(* IEC 61131-3 sources: SMRamp/src/Ar/SMRamp, 21 files *)

(* ---- SMRamp.typ ---- *)
(*
* File: SMRamp.typ
* Copyright (c) 2023 Loupe
* https://loupe.team
*
* This file is part of SMRamp, licensed under the MIT License.
*
*)

TYPE
	SMR_Axis_Int_ParUpdate_typ : 	STRUCT
		Update : BOOL;
		CurrValue : UINT;
		AccWrite : AsIOAccWrite;
	END_STRUCT;
	SMR_Axis_Int_Homing_typ : 	STRUCT
		State : UINT;
		CurrDirection : SINT; (*Current direction of travel*)
		HomeSwOld : BOOL; (*Previous value of HomeSw input for edge detection*)
		RisingEdge : BOOL; (*A rising edge was detected (not dependent on direction of travel)*)
		FallingEdge : BOOL; (*A falling edge was detected (not dependent on direction of travel)*)
		PosEdge : BOOL; (*A "Positive" edge was detected (depends on direction of travel)*)
		NegEdge : BOOL; (*A "Negative" edge was detected (depends on direction of travel)*)
		PosLimitSwOld : BOOL; (*Previous value of PosLimitSw for edge detection*)
		PosLimitSwRisingEdge : BOOL; (*An edge was detected for the PosLimitSw*)
		PosLimitSwFallingEdge : BOOL; (*An edge was detected for the PosLimitSw*)
		NegLimitSwOld : BOOL; (*Previous value of NegLimitSw for edge detection*)
		NegLimitSwRisingEdge : BOOL; (*An edge was detected for the NegLimitSw*)
		NegLimitSwFallingEdge : BOOL; (*An edge was detected for the NegLimitSw*)
		TargetReachedTimer : TON; (*Timer to ensure that TargetReached is true for long enough (takes care of timing issues, but makes homing slightly slower (100-200ms)).*)
	END_STRUCT;
	SMR_Axis_Internal_typ : 	STRUCT
		CMD : SMR_Axis_IN_CMD_typ; (*Internal CMD structure for discriminating between new and old commands.*)
		DIGIN : SMR_Axis_IOMap_IN_typ; (*Holds logical values of digital inputs (for future expansion)*)
		AbsPos : DINT;
		AbsPosActVal : DINT;
		CurrTargetPos : DINT;
		CurrTargetVel : DINT;
		CurrDirection : SINT;
		EnableState : UINT;
		SetState : UINT;
		Error : BOOL; (*Internal code error*)
		TargetReachedTimer : TON; (*Timer to ensure that TargetReached is true for long enough. Used to set Busy and Done in velocity mode.*)
		AckResetTimer : TON; (*Timer to ensure that the hardware fault acknowledge bits are high for long enough to be seen*)
		Homing : SMR_Axis_Int_Homing_typ;
		UpdateVel : SMR_Axis_Int_ParUpdate_typ;
		UpdateAcc : SMR_Axis_Int_ParUpdate_typ;
		UpdateDec : SMR_Axis_Int_ParUpdate_typ;
		ParsOK : BOOL; (*All motion parameters are up to date*)
		RTInfo : RTInfo; (*RTInfo block to get cycle time*)
		SpdEst : SpeedEst; (*SpdEst block to estimate speed*)
	END_STRUCT;
	SMR_Axis_IOMap_OUT_typ : 	STRUCT
		AbsPos : DINT;
		MpGenControl : UINT;
		MpGenMode : SINT;
	END_STRUCT;
	SMR_Axis_IOMap_IN_typ : 	STRUCT
		HomeSw : BOOL;
		PosLimitSw : BOOL;
		NegLimitSw : BOOL;
		QuickStop : BOOL;
		AbsPosActVal : DINT;
		MpGenStatus : UINT;
	END_STRUCT;
	SMR_Axis_IOMap_typ : 	STRUCT
		IN : SMR_Axis_IOMap_IN_typ;
		OUT : SMR_Axis_IOMap_OUT_typ;
	END_STRUCT;
	SMR_Axis_TEST_STAT_typ : 	STRUCT
		Busy : BOOL;
		Done : BOOL;
		Error : BOOL; (*Motor Fault or InternalError exists*)
		ErrorID : UINT;
		ErrorString : STRING[SMR_STRLEN_ERROR];
		ActualPosition : DINT;
		ActualVelocity : REAL; (*NOT IMPLEMENTED YET*)
		State : UINT;
		DriveFault : BOOL;
		VoltageEnabled : BOOL;
		HomingOk : BOOL;
	END_STRUCT;
	SMR_Axis_TEST_typ : 	STRUCT
		Enable : BOOL;
		CMD : SMR_Axis_IN_CMD_typ;
		PAR : SMR_Axis_IN_PAR_typ;
		STAT : SMR_Axis_TEST_STAT_typ;
	END_STRUCT;
	SMR_Axis_OUT_STAT_DriveStat_typ : 	STRUCT
		RdyToSwOn : BOOL;
		SwOn : BOOL;
		OpEnabled : BOOL;
		Fault : BOOL;
		VoltageEnabled : BOOL;
		QuickStop : BOOL;
		SwOnDisabled : BOOL;
		Warning : BOOL;
		Remote : BOOL;
		TargetReached : BOOL;
		IntLimitActive : BOOL;
		MotorLoad0 : BOOL;
		MotorLoad1 : BOOL;
		MotorLoad2 : BOOL;
		HomingOk : BOOL;
	END_STRUCT;
	SMR_Axis_OUT_STAT_typ : 	STRUCT
		ReadyForCMD : BOOL;
		Busy : BOOL;
		Done : BOOL;
		Error : BOOL; (*Motor Fault or InternalError exists*)
		ErrorID : UINT;
		ErrorString : STRING[SMR_STRLEN_ERROR];
		ErrorState : UINT;
		ActualPosition : DINT;
		ActualVelocity : REAL; (*Velocity in usteps/s or cts/s, depending on IN.CFG.ABRCtrSyncAsync. THIS WILL NOT MATCH VELOCITY INPUT BECAUSE OF DIFFERENT UNITS.*)
		DriveStatus : SMR_Axis_OUT_STAT_DriveStat_typ;
		State : UINT;
	END_STRUCT;
	SMR_Axis_OUT_typ : 	STRUCT
		STAT : SMR_Axis_OUT_STAT_typ;
	END_STRUCT;
	SMR_Axis_IN_CFG_SpdEst_typ : 	STRUCT
		tf : REAL;
		deadband : DINT;
		K : REAL;
	END_STRUCT;
	SMR_Axis_IN_CFG_typ : 	STRUCT
		DisableAcyclicWrite : BOOL;
		ModuleINADeviceName : STRING[80];
		MotorIndex : USINT;
		UnderCurrentDetection : BOOL;
		ABRCtrSyncAsync : BOOL;
		StallDetection : BOOL;
		InvertDirection : BOOL;
		SpeedEstimator : SMR_Axis_IN_CFG_SpdEst_typ;
	END_STRUCT;
	SMR_Axis_IN_PAR_typ : 	STRUCT
		HomingPosition : DINT;
		HomingMode : SINT;
		HomingVelocity : UINT;
		HomingStartDir : SINT;
		HomingEdgeSw : SINT;
		HomingTriggDir : SINT;
		Position : DINT;
		Direction : SINT;
		Velocity : UINT;
		Acceleration : UINT;
		Deceleration : UINT;
		JogVelocity : UINT;
		StopDeceleration : UINT;
	END_STRUCT;
	SMR_Axis_IN_CMD_typ : 	STRUCT
		Power : BOOL;
		Home : BOOL;
		MoveAbsolute : BOOL;
		MoveAdditive : BOOL;
		MoveVelocity : BOOL;
		JogForward : BOOL;
		JogReverse : BOOL;
		TrackSetPosition : BOOL;
		Stop : BOOL;
		AcknowledgeError : BOOL;
	END_STRUCT;
	SMR_Axis_IN_typ : 	STRUCT
		CMD : SMR_Axis_IN_CMD_typ;
		PAR : SMR_Axis_IN_PAR_typ;
		CFG : SMR_Axis_IN_CFG_typ;
	END_STRUCT;
	SMR_Axis_typ : 	STRUCT
		IN : SMR_Axis_IN_typ;
		OUT : SMR_Axis_OUT_typ;
		TEST : SMR_Axis_TEST_typ;
		IOMap : SMR_Axis_IOMap_typ;
		Internal : SMR_Axis_Internal_typ;
	END_STRUCT;
END_TYPE

(* ---- SMR_CheckHomePAR.st ---- *)
(*
* File: SMR_CheckHomePAR.st
* Copyright (c) 2023 Loupe
* https://loupe.team
*
* This file is part of SMRamp, licensed under the MIT License.
*
*)

(*Function which checks homing parameters.  Returns TRUE if pars are OK.*)

(* Parameter checking			DONE and TESTED DFB 20090914 *)

FUNCTION SMR_CheckHomePAR

(* Reset internal Error variable.  Will be set below if there is an error *)

Error:=	0;

(* Check HomingMode *)

IF( 	(pAxis.IN.PAR.HomingMode <> SMR_HOMEMODE_DIRECT)
	AND (pAxis.IN.PAR.HomingMode <> SMR_HOMEMODE_SWITCH_GATE)
	AND	(pAxis.IN.PAR.HomingMode <> SMR_HOMEMODE_ABS_SWITCH)
	AND	(pAxis.IN.PAR.HomingMode <> SMR_HOMEMODE_END_SWITCH)
	)THEN

 	Error:=	1;

END_IF

(* Check HomingVelocity *)

IF( pAxis.IN.PAR.HomingVelocity = 0 )THEN

 	Error:=	1;

END_IF

(* Check HomingStartDir *)

IF( 	(pAxis.IN.PAR.HomingStartDir <> SMR_POS)
	AND (pAxis.IN.PAR.HomingStartDir <> SMR_NEG)
	)THEN

 	Error:=	1;

END_IF

(* Check HomingEdgeSw *)

IF( 	(pAxis.IN.PAR.HomingEdgeSw <> SMR_POS)
	AND	(pAxis.IN.PAR.HomingEdgeSw <> SMR_NEG)
	)THEN

 	Error:=	1;

END_IF

(* Check HomingTriggDir *)

IF( 	(pAxis.IN.PAR.HomingTriggDir <> SMR_POS)
	AND	(pAxis.IN.PAR.HomingTriggDir <> SMR_NEG)
	)THEN

 	Error:=	1;

END_IF

IF( Error )THEN

	SMR_CheckHomePAR:=	0;

ELSE

	SMR_CheckHomePAR:=	1;

END_IF

END_FUNCTION

(* ---- SMR_CheckLimitSw.st ---- *)
(*
* File: SMR_CheckLimitSw.st
* Copyright (c) 2023 Loupe
* https://loupe.team
*
* This file is part of SMRamp, licensed under the MIT License.
*
*)

(********************************************************************)
(* Check limit switches 											*)
(********************************************************************)

FUNCTION SMR_CheckLimitSw

(********************************************************************)
(* Set return value to get rid of compiler warning					*)
(********************************************************************)

SMR_CheckLimitSw:=	FALSE;

(********************************************************************)
(* Check Limit Switches												*)
(********************************************************************)

(* PosLimitSw *)

IF( (pAxis.Internal.CurrDirection = SMR_DIR_POS)
	AND	(pAxis.Internal.DIGIN.PosLimitSw)
	)THEN

	(* Set CurrDirection to STOP *)

	pAxis.Internal.CurrDirection:=	SMR_DIR_STOP;

	(* Set Mode to Velocity mode and set position to 0 to stop axis *)

	pAxis.IOMap.OUT.MpGenMode:=	SMR_MODE_VELOCITY;
	pAxis.Internal.AbsPos:=		0;

	(* Set Error info and go to Error state *)

	pAxis.Internal.Error:=			1;
	pAxis.OUT.STAT.ErrorID:=		SMR_ERR_POSLIMSW;
	pAxis.OUT.STAT.ErrorState:=		pAxis.Internal.EnableState;

	pAxis.Internal.EnableState:=	SMR_STEN_ERROR;

	(* Reset Busy and Done *)

	pAxis.OUT.STAT.Busy:=	0;
	pAxis.OUT.STAT.Done:=	0;

END_IF

(* NegLimitSw *)

IF( (pAxis.Internal.CurrDirection = SMR_DIR_NEG)
	AND	(pAxis.Internal.DIGIN.NegLimitSw)
	)THEN

	(* Set CurrDirection to STOP *)

	pAxis.Internal.CurrDirection:=	SMR_DIR_STOP;

	(* Set Mode to Velocity mode and set position to 0 to stop axis *)

	pAxis.IOMap.OUT.MpGenMode:=	SMR_MODE_VELOCITY;
	pAxis.Internal.AbsPos:=		0;

	(* Set Error info and go to Error state *)

	pAxis.Internal.Error:=			1;
	pAxis.OUT.STAT.ErrorID:=		SMR_ERR_NEGLIMSW;
	pAxis.OUT.STAT.ErrorState:=		pAxis.Internal.EnableState;

	pAxis.Internal.EnableState:=	SMR_STEN_ERROR;

	(* Reset Busy and Done *)

	pAxis.OUT.STAT.Busy:=	0;
	pAxis.OUT.STAT.Done:=	0;

END_IF

END_FUNCTION

(* ---- SMR_GetDriveStatus.st ---- *)
(*
* File: SMR_GetDriveStatus.st
* Copyright (c) 2023 Loupe
* https://loupe.team
*
* This file is part of SMRamp, licensed under the MIT License.
*
*)

(*This is an internal function that maps out the status from the status UINT.*)

(* Getting status			DONE and TESTED DFB 20110329 *)

FUNCTION SMR_GetDriveStatus

(********************************************************************)
(* Set return value to get rid of compiler warning					*)
(********************************************************************)

SMR_GetDriveStatus:=	FALSE;

(* Get status BOOLs out of status UINT *)

DriveStatus.RdyToSwOn:=			BIT_TST(MpGenStatus, 0);
DriveStatus.SwOn:=				BIT_TST(MpGenStatus, 1);
DriveStatus.OpEnabled:=			BIT_TST(MpGenStatus, 2);
DriveStatus.Fault:=				BIT_TST(MpGenStatus, 3);
DriveStatus.VoltageEnabled:=	BIT_TST(MpGenStatus, 4);
DriveStatus.QuickStop:=			BIT_TST(MpGenStatus, 5);
DriveStatus.SwOnDisabled:=		BIT_TST(MpGenStatus, 6);
DriveStatus.Warning:=			BIT_TST(MpGenStatus, 7);

DriveStatus.Remote:=			BIT_TST(MpGenStatus, 9);
DriveStatus.TargetReached:=		BIT_TST(MpGenStatus, 10);
DriveStatus.IntLimitActive:=	BIT_TST(MpGenStatus, 11);

DriveStatus.MotorLoad0:=		BIT_TST(MpGenStatus, 13);
DriveStatus.MotorLoad1:=		BIT_TST(MpGenStatus, 14);
DriveStatus.MotorLoad2:=		BIT_TST(MpGenStatus, 15);

END_FUNCTION

(* ---- SMR_Home.st ---- *)
(*
* File: SMR_Home.st
* Copyright (c) 2023 Loupe
* https://loupe.team
*
* This file is part of SMRamp, licensed under the MIT License.
*
*)

(*Function to perform homing functionality.*)

(* Stop during home										DONE and TESTED DFB 20110404 *)
	(* Setting SetState									DONE and TESTED DFB 20110404 *)
	(* Changing State									DONE and TESTED DFB 20110404 *)

(* Checking parameters									see CheckHomePAR.st *)
	(* Finding bad parameters							see CheckHomePAR.st *)
	(* Reacting to bad parameters						DONE and TESTED DFB 20090918 *)

(* Finding events										see HomeFindEdge.st *)

(* Starting Homing - change state based on mode			DONE and TESTED DFB 20090918 *)

(* Homing Modes											DONE and TESTED DFB 20090921 *)

	(* Direct											DONE and TESTED DFB 20090918 *)

	(* Switch gate mode									DONE and TESTED DFB 20090918 *)

		(* StartDir = Positive							DONE and TESTED DFB 20090918 *)

			(* EdgeSw = Positive						DONE and TESTED DFB 20090918 *)
				(* TriggDir = Positive					DONE and TESTED DFB 20090918 *)
				(* TriggDir = Negative					DONE and TESTED DFB 20090918 *)

			(* EdgeSw = Negative						DONE and TESTED DFB 20090918 *)
				(* TriggDir = Positive					DONE and TESTED DFB 20090918 *)
				(* TriggDir = Negative					DONE and TESTED DFB 20090918 *)

		(* StartDir = Negative							DONE and TESTED DFB 20090918 *)

			(* EdgeSw = Positive						DONE and TESTED DFB 20090918 *)
				(* TriggDir = Positive					DONE and TESTED DFB 20090918 *)
				(* TriggDir = Negative					DONE and TESTED DFB 20090918 *)

			(* EdgeSw = Negative						DONE and TESTED DFB 20090918 *)
				(* TriggDir = Positive					DONE and TESTED DFB 20090918 *)
				(* TriggDir = Negative					DONE and TESTED DFB 20090918 *)

	(* Abs Switch mode									DONE and TESTED DFB 20090918 *)

		(* EdgeSw = Positive							DONE and TESTED DFB 20090918 *)
			(* TriggDir = Positive						DONE and TESTED DFB 20090918 *)
			(* TriggDir = Negative						DONE and TESTED DFB 20090918 *)

		(* EdgeSw = Negative							DONE and TESTED DFB 20090918 *)
			(* TriggDir = Positive						DONE and TESTED DFB 20090918 *)
			(* TriggDir = Negative						DONE and TESTED DFB 20090918 *)

	(* End switch										DONE and TESTED DFB 20090921 *)

		(* EdgeSw = Positive							DONE and TESTED DFB 20090921 *)
			(* TriggDir = Positive						DONE and TESTED DFB 20090921 *)
			(* TriggDir = Negative						DONE and TESTED DFB 20090921 *)

		(* EdgeSw = Negative							DONE and TESTED DFB 20090921 *)
			(* TriggDir = Positive						DONE and TESTED DFB 20090921 *)
			(* TriggDir = Negative						DONE and TESTED DFB 20090921 *)

(* Finishing homing										DONE and TESTED DFB 20090918 *)

	(* Setting ActPos to HomeOffset						DONE and TESTED DFB 20090918 *)
		(* Mode and AbsPos setting						DONE and TESTED DFB 20110906 *)

	(* Timing on TargetReached							DONE and TESTED DFB 20090918 *)
		(* 5ms TC										DONE and TESTED DFB 20090918 *)
		(* 25ms TC										DONE and TESTED DFB 20090918 *)
		(* 50ms TC										DONE and TESTED DFB 20090918 *)

	(* Being at HomeOffset after homing					DONE and TESTED DFB 20090918 *)
		(* Mode and AbsPos setting						DONE and TESTED DFB 20110906 *)

	(* Setting HomingComplete 							DONE and TESTED DFB 20090918 *)

FUNCTION SMR_Home

(********************************************************************)
(* Set return value to get rid of compiler warning					*)
(********************************************************************)

SMR_Home:=	FALSE;

(* Map pointer to internal homing variables *)

t ACCESS ADR(pAxis.Internal.Homing);

(********************************************************************)
(* Reset TargetReachedTimer.  It will be set below when appropriate	*)
(********************************************************************)

t.TargetReachedTimer.IN:=	0;

(********************************************************************)
(* Stop command can interrupt a home move 							*)
(********************************************************************)

IF( pAxis.IN.CMD.Stop ) THEN

	(* Set the target state as SETSTOP *)

	pAxis.Internal.SetState:=		SMR_STEN_SETSTOP;

	(* Set Busy, Done *)

	pAxis.OUT.STAT.Busy:=	1;
	pAxis.OUT.STAT.Done:=	0;

	(* Go to SetState *)

	pAxis.Internal.EnableState:=	pAxis.Internal.SetState;

	RETURN;

END_IF

(********************************************************************)
(* Check Homing Parameters											*)
(********************************************************************)

IF( SMR_CheckHomePAR( pAxis ) = FALSE ) THEN

	(* Error - set internal error and go to error state *)

	pAxis.Internal.Error:=			1;
	pAxis.OUT.STAT.ErrorID:=		SMR_ERR_HOME_INVALIDPAR;
	pAxis.OUT.STAT.ErrorState:=		pAxis.Internal.EnableState;

	pAxis.Internal.EnableState:=	SMR_STEN_ERROR;

	RETURN;

END_IF

(********************************************************************)
(* Find edges 														*)
(********************************************************************)

SMR_HomeFindEdge( pAxis );

(********************************************************************)
(* Main State Machine												*)
(********************************************************************)

CASE t.State OF

	(********************************************************************)
	(* Starting Homing													*)
	(********************************************************************)

	SMR_STHOME_CHECKMODE:

		(* Stop motor when homing is initiated *)

		pAxis.IOMap.OUT.MpGenMode:=	SMR_MODE_VELOCITY;
		pAxis.Internal.AbsPos:=		0;

		(* Change state based on homing mode *)

		IF( pAxis.IN.PAR.HomingMode = SMR_HOMEMODE_DIRECT ) THEN

			(* If direct home, set homeoffset directly after motor is stopped *)

			t.State:=	SMR_STHOME_STOPPING;

  		ELSIF( pAxis.IN.PAR.HomingMode = SMR_HOMEMODE_SWITCH_GATE ) THEN

			t.State:=	SMR_STHOME_SG_START;

  		ELSIF( pAxis.IN.PAR.HomingMode = SMR_HOMEMODE_ABS_SWITCH ) THEN

			t.State:=	SMR_STHOME_ABS_START;

  		ELSIF( pAxis.IN.PAR.HomingMode = SMR_HOMEMODE_END_SWITCH ) THEN

			t.State:=	SMR_STHOME_END_START;

		END_IF

	(********************************************************************)
	(* Switch Gate mode													*)
	(********************************************************************)

	SMR_STHOME_SG_START:

		IF( pAxis.IN.PAR.HomingStartDir = SMR_POS ) THEN

			IF( pAxis.Internal.DIGIN.PosLimitSw ) THEN

   				t.CurrDirection:=	SMR_DIR_NEG;

			ELSE

				t.CurrDirection:=	SMR_DIR_POS;

			END_IF

		ELSIF( pAxis.IN.PAR.HomingStartDir = SMR_NEG ) THEN

			IF( pAxis.Internal.DIGIN.NegLimitSw ) THEN

   				t.CurrDirection:=	SMR_DIR_POS;

			ELSE

				t.CurrDirection:=	SMR_DIR_NEG;

			END_IF

		END_IF

		(* Change state *)

		t.State:=	SMR_STHOME_SG_MOVE;

		(* Set mode and velocity *)

		pAxis.IOMap.OUT.MpGenMode:=	SMR_MODE_VELOCITY;
		pAxis.Internal.AbsPos:=		UINT_TO_DINT(pAxis.IN.PAR.HomingVelocity) * t.CurrDirection;

	SMR_STHOME_SG_MOVE:

		(* Check all possible events and react accordingly *)

		(****************************************************)
		(* NegLimitSw *)

		IF( pAxis.Internal.DIGIN.NegLimitSw ) THEN

			(************************************************)
			(* NegLimitSw, NegDir *)

			IF( t.CurrDirection = SMR_DIR_NEG ) THEN

   				IF( pAxis.IN.PAR.HomingStartDir = SMR_POS ) THEN

					(* Stop, error *)

					t.CurrDirection:=	SMR_DIR_STOP;

					pAxis.Internal.Error:=			1;
					pAxis.OUT.STAT.ErrorID:=		SMR_ERR_HOME_ERR;
					pAxis.OUT.STAT.ErrorState:=		pAxis.Internal.EnableState;

					pAxis.Internal.EnableState:=	SMR_STEN_ERROR;

	   			ELSIF( pAxis.IN.PAR.HomingStartDir = SMR_NEG ) THEN

					(* Turn around to look for switch *)

					t.CurrDirection:=	SMR_DIR_POS;

				END_IF (* HomeStartDir *)

   			END_IF (* CurrDirection *)

		(****************************************************)
		(* PosLimitSw *)

		ELSIF( pAxis.Internal.DIGIN.PosLimitSw ) THEN

			(************************************************)
			(* PosLimitSw, PosDir *)

			IF( t.CurrDirection = SMR_DIR_POS ) THEN

				IF( pAxis.IN.PAR.HomingStartDir = SMR_POS ) THEN

					(* Turn around to look for switch *)

					t.CurrDirection:=	SMR_DIR_NEG;

	   			ELSIF( pAxis.IN.PAR.HomingStartDir = SMR_NEG ) THEN

					(* Stop, error *)

					t.CurrDirection:=	SMR_DIR_STOP;

					pAxis.Internal.Error:=			1;
					pAxis.OUT.STAT.ErrorID:=		SMR_ERR_HOME_ERR;
					pAxis.OUT.STAT.ErrorState:=		pAxis.Internal.EnableState;

					pAxis.Internal.EnableState:=	SMR_STEN_ERROR;

				END_IF (* HomeStartDir *)

			END_IF (* CurrDirection *)

		(****************************************************)
		(* PosEdge *)

		ELSIF( t.PosEdge ) THEN

  			(************************************************)
			(* PosEdge, PosDir *)

			IF( t.CurrDirection = SMR_DIR_POS ) THEN

				IF( pAxis.IN.PAR.HomingEdgeSw = SMR_POS ) THEN

					IF( pAxis.IN.PAR.HomingTriggDir = SMR_POS ) THEN

						(* Stop, done *)

						t.CurrDirection:=	SMR_DIR_STOP;

						t.State:=			SMR_STHOME_STOPPING;

	 				ELSIF( pAxis.IN.PAR.HomingTriggDir = SMR_NEG ) THEN

						(* Go negative *)

						t.CurrDirection:=	SMR_DIR_NEG;

	 				END_IF (* HomeTriggDir *)

				ELSIF( pAxis.IN.PAR.HomingEdgeSw = SMR_NEG ) THEN

					(* Find negative edge *)

					t.CurrDirection:=	SMR_DIR_POS;

				END_IF (* HomeEdgeSw *)

   			(************************************************)
			(* PosEdge, NegDir *)

			ELSIF( t.CurrDirection = SMR_DIR_NEG ) THEN

				IF( pAxis.IN.PAR.HomingEdgeSw = SMR_POS ) THEN

					IF( pAxis.IN.PAR.HomingTriggDir = SMR_POS ) THEN

						(* Go positive *)

						t.CurrDirection:=	SMR_DIR_POS;

	 				ELSIF( pAxis.IN.PAR.HomingTriggDir = SMR_NEG ) THEN

						(* Stop, done *)

						t.CurrDirection:=	SMR_DIR_STOP;

						t.State:=			SMR_STHOME_STOPPING;

	 				END_IF (* HomeTriggDir *)

				ELSIF( pAxis.IN.PAR.HomingEdgeSw = SMR_NEG ) THEN

					(* Find negative edge *)

					t.CurrDirection:=	SMR_DIR_POS;

				END_IF (* HomeEdgeSw *)

   			END_IF (* CurrDirection *)

		(****************************************************)
		(* NegEdge *)

  		ELSIF( t.NegEdge ) THEN

  			(************************************************)
			(* NegEdge, PosDir *)

			IF( t.CurrDirection = SMR_DIR_POS ) THEN

				IF( pAxis.IN.PAR.HomingEdgeSw = SMR_POS ) THEN

					(* Find positive edge *)

					t.CurrDirection:=	SMR_DIR_NEG;

				ELSIF( pAxis.IN.PAR.HomingEdgeSw = SMR_NEG ) THEN

					IF( pAxis.IN.PAR.HomingTriggDir = SMR_POS ) THEN

						(* Stop, done *)

						t.CurrDirection:=	SMR_DIR_STOP;

						t.State:=			SMR_STHOME_STOPPING;

	 				ELSIF( pAxis.IN.PAR.HomingTriggDir = SMR_NEG ) THEN

						(* Go negative *)

						t.CurrDirection:=	SMR_DIR_NEG;

	 				END_IF (* HomeTriggDir *)

				END_IF (* HomeEdgeSw *)

   			(************************************************)
			(* NegEdge, NegDir *)

			ELSIF( t.CurrDirection = SMR_DIR_NEG ) THEN

				IF( pAxis.IN.PAR.HomingEdgeSw = SMR_POS ) THEN

					(* Find positive edge *)

					t.CurrDirection:=	SMR_DIR_NEG;

				ELSIF( pAxis.IN.PAR.HomingEdgeSw = SMR_NEG ) THEN

					IF( pAxis.IN.PAR.HomingTriggDir = SMR_POS ) THEN

						(* Go positive *)

						t.CurrDirection:=	SMR_DIR_POS;

	 				ELSIF( pAxis.IN.PAR.HomingTriggDir = SMR_NEG ) THEN

						(* Stop, done *)

						t.CurrDirection:=	SMR_DIR_STOP;

						t.State:=			SMR_STHOME_STOPPING;

	 				END_IF (* HomeTriggDir *)

				END_IF (* HomeEdgeSw *)

   			END_IF (* CurrDirection *)

  		END_IF (* Events *)

		(* Set mode and velocity *)

		pAxis.IOMap.OUT.MpGenMode:=	SMR_MODE_VELOCITY;
		pAxis.Internal.AbsPos:=		UINT_TO_DINT(pAxis.IN.PAR.HomingVelocity) * t.CurrDirection;

	(********************************************************************)
	(* Absolute Switch mode												*)
	(********************************************************************)

	SMR_STHOME_ABS_START:

		(* Start based on EdgeSw and current level of switch *)

		IF( pAxis.IN.PAR.HomingEdgeSw = SMR_POS ) THEN

			IF( pAxis.Internal.DIGIN.HomeSw ) THEN

   				t.CurrDirection:=	SMR_DIR_NEG;

   			ELSE

				t.CurrDirection:=	SMR_DIR_POS;

			END_IF (* HomeSw *)

		ELSIF( pAxis.IN.PAR.HomingEdgeSw = SMR_NEG ) THEN

			IF( pAxis.Internal.DIGIN.HomeSw ) THEN

   				t.CurrDirection:=	SMR_DIR_POS;

   			ELSE

				t.CurrDirection:=	SMR_DIR_NEG;

			END_IF (* HomeSw *)

		END_IF (* HomeEdgeSw *)

		(* Change state *)

		t.State:=	SMR_STHOME_ABS_MOVE;

		(* Set mode and velocity *)

		pAxis.IOMap.OUT.MpGenMode:=	SMR_MODE_VELOCITY;
		pAxis.Internal.AbsPos:=		UINT_TO_DINT(pAxis.IN.PAR.HomingVelocity) * t.CurrDirection;

	SMR_STHOME_ABS_MOVE:

		(* Check all possible events and react accordingly *)

		(****************************************************)
		(* NegLimitSw, Negative Dir *)

		IF( (pAxis.Internal.DIGIN.NegLimitSw)	AND
  			(t.CurrDirection = SMR_DIR_NEG)		) THEN

			(* Stop, error *)

			t.CurrDirection:=	SMR_DIR_STOP;

			pAxis.Internal.Error:=			1;
			pAxis.OUT.STAT.ErrorID:=		SMR_ERR_HOME_ERR;
			pAxis.OUT.STAT.ErrorState:=		pAxis.Internal.EnableState;

			pAxis.Internal.EnableState:=	SMR_STEN_ERROR;

		(****************************************************)
		(* PosLimitSw, Positive Dir *)

		ELSIF(	(pAxis.Internal.DIGIN.PosLimitSw)	AND
	  			(t.CurrDirection = SMR_DIR_POS)		) THEN

			(* Stop, error *)

			t.CurrDirection:=	SMR_DIR_STOP;

			pAxis.Internal.Error:=			1;
			pAxis.OUT.STAT.ErrorID:=		SMR_ERR_HOME_ERR;
			pAxis.OUT.STAT.ErrorState:=		pAxis.Internal.EnableState;

			pAxis.Internal.EnableState:=	SMR_STEN_ERROR;

		(****************************************************)
		(* PosEdge *)

		ELSIF( t.PosEdge ) THEN

  			(************************************************)
			(* PosEdge, PosDir *)

			IF( t.CurrDirection = SMR_DIR_POS ) THEN

				IF( pAxis.IN.PAR.HomingEdgeSw = SMR_POS ) THEN

					IF( pAxis.IN.PAR.HomingTriggDir = SMR_POS ) THEN

						(* Stop, done *)

						t.CurrDirection:=	SMR_DIR_STOP;

						t.State:=			SMR_STHOME_STOPPING;

	 				ELSIF( pAxis.IN.PAR.HomingTriggDir = SMR_NEG ) THEN

						(* Go negative *)

						t.CurrDirection:=	SMR_DIR_NEG;

	 				END_IF (* HomeTriggDir *)

				ELSIF( pAxis.IN.PAR.HomingEdgeSw = SMR_NEG ) THEN

					(* Stop, error *)

					t.CurrDirection:=	SMR_DIR_STOP;

					pAxis.Internal.Error:=			1;
					pAxis.OUT.STAT.ErrorID:=		SMR_ERR_HOME_ERR;
					pAxis.OUT.STAT.ErrorState:=		pAxis.Internal.EnableState;

					pAxis.Internal.EnableState:=	SMR_STEN_ERROR;

				END_IF (* HomeEdgeSw *)

   			(************************************************)
			(* PosEdge, NegDir *)

			ELSIF( t.CurrDirection = SMR_DIR_NEG ) THEN

				IF( pAxis.IN.PAR.HomingEdgeSw = SMR_POS ) THEN

					IF( pAxis.IN.PAR.HomingTriggDir = SMR_POS ) THEN

						(* Go positive *)

						t.CurrDirection:=	SMR_DIR_POS;

	 				ELSIF( pAxis.IN.PAR.HomingTriggDir = SMR_NEG ) THEN

						(* Stop, done *)

						t.CurrDirection:=	SMR_DIR_STOP;

						t.State:=			SMR_STHOME_STOPPING;

	 				END_IF (* HomeTriggDir *)

				ELSIF( pAxis.IN.PAR.HomingEdgeSw = SMR_NEG ) THEN

					(* Stop, error *)

					t.CurrDirection:=	SMR_DIR_STOP;

					pAxis.Internal.Error:=			1;
					pAxis.OUT.STAT.ErrorID:=		SMR_ERR_HOME_ERR;
					pAxis.OUT.STAT.ErrorState:=		pAxis.Internal.EnableState;

					pAxis.Internal.EnableState:=	SMR_STEN_ERROR;

				END_IF (* HomeEdgeSw *)

   			END_IF (* CurrDirection *)

		(****************************************************)
		(* NegEdge *)

  		ELSIF( t.NegEdge ) THEN

  			(************************************************)
			(* NegEdge, PosDir *)

			IF( t.CurrDirection = SMR_DIR_POS ) THEN

				IF( pAxis.IN.PAR.HomingEdgeSw = SMR_POS ) THEN

					(* Stop, error *)

					t.CurrDirection:=	SMR_DIR_STOP;

					pAxis.Internal.Error:=			1;
					pAxis.OUT.STAT.ErrorID:=		SMR_ERR_HOME_ERR;
					pAxis.OUT.STAT.ErrorState:=		pAxis.Internal.EnableState;

					pAxis.Internal.EnableState:=	SMR_STEN_ERROR;

				ELSIF( pAxis.IN.PAR.HomingEdgeSw = SMR_NEG ) THEN

					IF( pAxis.IN.PAR.HomingTriggDir = SMR_POS ) THEN

						(* Stop, done *)

						t.CurrDirection:=	SMR_DIR_STOP;

						t.State:=			SMR_STHOME_STOPPING;

	 				ELSIF( pAxis.IN.PAR.HomingTriggDir = SMR_NEG ) THEN

						(* Go negative *)

						t.CurrDirection:=	SMR_DIR_NEG;

	 				END_IF (* HomeTriggDir *)

				END_IF (* HomeEdgeSw *)

   			(************************************************)
			(* NegEdge, NegDir *)

			ELSIF( t.CurrDirection = SMR_DIR_NEG ) THEN

				IF( pAxis.IN.PAR.HomingEdgeSw = SMR_POS ) THEN

					(* Stop, error *)

					t.CurrDirection:=	SMR_DIR_STOP;

					pAxis.Internal.Error:=			1;
					pAxis.OUT.STAT.ErrorID:=		SMR_ERR_HOME_ERR;
					pAxis.OUT.STAT.ErrorState:=		pAxis.Internal.EnableState;

					pAxis.Internal.EnableState:=	SMR_STEN_ERROR;

				ELSIF( pAxis.IN.PAR.HomingEdgeSw = SMR_NEG ) THEN

					IF( pAxis.IN.PAR.HomingTriggDir = SMR_POS ) THEN

						(* Go positive *)

						t.CurrDirection:=	SMR_DIR_POS;

	 				ELSIF( pAxis.IN.PAR.HomingTriggDir = SMR_NEG ) THEN

						(* Stop, done *)

						t.CurrDirection:=	SMR_DIR_STOP;

						t.State:=			SMR_STHOME_STOPPING;

	 				END_IF (* HomeTriggDir *)

				END_IF (* HomeEdgeSw *)

   			END_IF (* CurrDirection *)

  		END_IF (* Events *)

		(* Set mode and velocity *)

		pAxis.IOMap.OUT.MpGenMode:=	SMR_MODE_VELOCITY;
		pAxis.Internal.AbsPos:=		UINT_TO_DINT(pAxis.IN.PAR.HomingVelocity) * t.CurrDirection;

	(********************************************************************)
	(* End (Limit) Switch mode											*)
	(********************************************************************)

	SMR_STHOME_END_START:

		(* Start based on EdgeSw and current level of switches *)

		IF( pAxis.IN.PAR.HomingEdgeSw = SMR_POS ) THEN

			IF( pAxis.Internal.DIGIN.PosLimitSw ) THEN

   				t.CurrDirection:=	SMR_DIR_NEG;

   			ELSE

				t.CurrDirection:=	SMR_DIR_POS;

			END_IF (* PosLimitSw *)

		ELSIF( pAxis.IN.PAR.HomingEdgeSw = SMR_NEG ) THEN

			IF( pAxis.Internal.DIGIN.NegLimitSw ) THEN

   				t.CurrDirection:=	SMR_DIR_POS;

   			ELSE

				t.CurrDirection:=	SMR_DIR_NEG;

			END_IF (* NegLimitSw *)

		END_IF (* HomeEdgeSw *)

		(* Change state *)

		t.State:=	SMR_STHOME_END_MOVE;

		(* Set mode and velocity *)

		pAxis.IOMap.OUT.MpGenMode:=	SMR_MODE_VELOCITY;
		pAxis.Internal.AbsPos:=		UINT_TO_DINT(pAxis.IN.PAR.HomingVelocity) * t.CurrDirection;

	SMR_STHOME_END_MOVE:

		(* Check events and react accordingly *)

		IF( t.PosLimitSwRisingEdge ) THEN

			IF( pAxis.IN.PAR.HomingEdgeSw = SMR_POS ) THEN

				IF( pAxis.IN.PAR.HomingTriggDir = SMR_POS ) THEN

					(* Stop, done *)

					t.CurrDirection:=	SMR_DIR_STOP;

					t.State:=			SMR_STHOME_STOPPING;

				ELSIF( pAxis.IN.PAR.HomingTriggDir = SMR_NEG ) THEN

					(* go neg until you see a falling edge *)

					t.CurrDirection:=	SMR_DIR_NEG;

	   			END_IF (* HomeTriggDir *)

	  		ELSIF( pAxis.IN.PAR.HomingEdgeSw = SMR_NEG ) THEN

				(* Stop, error *)

				t.CurrDirection:=	SMR_DIR_STOP;

				pAxis.Internal.Error:=			1;
				pAxis.OUT.STAT.ErrorID:=		SMR_ERR_HOME_ERR;
				pAxis.OUT.STAT.ErrorState:=		pAxis.Internal.EnableState;

				pAxis.Internal.EnableState:=	SMR_STEN_ERROR;

			END_IF (* HomeEdgeSw *)

		ELSIF( t.PosLimitSwFallingEdge ) THEN

			IF( pAxis.IN.PAR.HomingEdgeSw = SMR_POS ) THEN

				IF( pAxis.IN.PAR.HomingTriggDir = SMR_POS ) THEN

					(* go pos until you see a rising edge *)

					t.CurrDirection:=	SMR_DIR_POS;

				ELSIF( pAxis.IN.PAR.HomingTriggDir = SMR_NEG ) THEN

					(* Stop, done *)

					t.CurrDirection:=	SMR_DIR_STOP;

					t.State:=			SMR_STHOME_STOPPING;

	   			END_IF (* HomeTriggDir *)

	  		ELSIF( pAxis.IN.PAR.HomingEdgeSw = SMR_NEG ) THEN

				(* Continue in negative direction *)

				t.CurrDirection:=	SMR_DIR_NEG;

			END_IF (* HomeEdgeSw *)

		ELSIF( t.NegLimitSwRisingEdge ) THEN

			IF( pAxis.IN.PAR.HomingEdgeSw = SMR_POS ) THEN

				(* Stop, error *)

				t.CurrDirection:=	SMR_DIR_STOP;

				pAxis.Internal.Error:=			1;
				pAxis.OUT.STAT.ErrorID:=		SMR_ERR_HOME_ERR;
				pAxis.OUT.STAT.ErrorState:=		pAxis.Internal.EnableState;

				pAxis.Internal.EnableState:=	SMR_STEN_ERROR;

	  		ELSIF( pAxis.IN.PAR.HomingEdgeSw = SMR_NEG ) THEN

				IF( pAxis.IN.PAR.HomingTriggDir = SMR_POS ) THEN

					(* go pos until you see a falling edge *)

					t.CurrDirection:=	SMR_DIR_POS;

				ELSIF( pAxis.IN.PAR.HomingTriggDir = SMR_NEG ) THEN

					(* Stop, done *)

					t.CurrDirection:=	SMR_DIR_STOP;

					t.State:=			SMR_STHOME_STOPPING;

	   			END_IF (* HomeTriggDir *)

			END_IF (* HomeEdgeSw *)

		ELSIF( t.NegLimitSwFallingEdge ) THEN

			IF( pAxis.IN.PAR.HomingEdgeSw = SMR_POS ) THEN

				(* Continue in positive direction *)

				t.CurrDirection:=	SMR_DIR_POS;

	  		ELSIF( pAxis.IN.PAR.HomingEdgeSw = SMR_NEG ) THEN

				IF( pAxis.IN.PAR.HomingTriggDir = SMR_POS ) THEN

					(* Stop, done *)

					t.CurrDirection:=	SMR_DIR_STOP;

					t.State:=			SMR_STHOME_STOPPING;

				ELSIF( pAxis.IN.PAR.HomingTriggDir = SMR_NEG ) THEN

					(* go neg until you see a rising edge *)

					t.CurrDirection:=	SMR_DIR_NEG;

	   			END_IF (* HomeTriggDir *)

			END_IF (* HomeEdgeSw *)

		END_IF (* Events *)

		(* Set mode and velocity *)

		pAxis.IOMap.OUT.MpGenMode:=	SMR_MODE_VELOCITY;
		pAxis.Internal.AbsPos:=		UINT_TO_DINT(pAxis.IN.PAR.HomingVelocity) * t.CurrDirection;

	(********************************************************************)
	(* Finishing Homing													*)
	(********************************************************************)

	SMR_STHOME_STOPPING:

		(* If TargetReached, start the timer *)

		t.TargetReachedTimer.IN:=	pAxis.OUT.STAT.DriveStatus.TargetReached;

		(* If the timer expires, then TargetReached is real, not just a blip *)

		IF( t.TargetReachedTimer.Q ) THEN

			(* Reset timer for next state to use *)

			t.TargetReachedTimer.IN:=	0;

			(* If TargetReached, set current position to HomingPosition *)

			pAxis.IOMap.OUT.MpGenMode:=	SMR_MODE_SETACTPOS;
			pAxis.Internal.AbsPos:=		pAxis.IN.PAR.HomingPosition;

			t.State:=	SMR_STHOME_DONE;

		END_IF

	SMR_STHOME_DONE:

		(* If TargetReached, start the timer *)

		t.TargetReachedTimer.IN:=	pAxis.OUT.STAT.DriveStatus.TargetReached;

		(* If the timer expires, then TargetReached is real, not just a blip *)

		IF( t.TargetReachedTimer.Q ) THEN

			(* Reset timer for next state to use *)

			t.TargetReachedTimer.IN:=	0;

			(* If TargetReached, change to position mode, move to HomingPosition, and return to wait state *)

			pAxis.OUT.STAT.DriveStatus.HomingOk:=	1;

			pAxis.IOMap.OUT.MpGenMode:=		SMR_MODE_POSITION;
			pAxis.Internal.AbsPos:=			pAxis.IN.PAR.HomingPosition;
			pAxis.Internal.CurrTargetPos:=	pAxis.IN.PAR.HomingPosition;

			(* Return to wait state *)

			pAxis.Internal.EnableState:=	SMR_STEN_WAIT;

		END_IF

END_CASE

(********************************************************************)
(* Call Timer FUB													*)
(********************************************************************)

t.TargetReachedTimer.PT:=	T#50ms;
t.TargetReachedTimer();

END_FUNCTION

(* ---- SMR_HomeFindEdge.st ---- *)
(*
* File: SMR_HomeFindEdge.st
* Copyright (c) 2023 Loupe
* https://loupe.team
*
* This file is part of SMRamp, licensed under the MIT License.
*
*)

(*Function to find edges for homing.*)

(* Rising edges			DONE and TESTED DFB 20090914 *)
(* Falling edges		DONE and TESTED DFB 20090914 *)

(* Positive edges		DONE and TESTED DFB 20090914 *)
(* Negative edges		DONE and TESTED DFB 20090914 *)

(* PosLimitSw edges		DONE and TESTED DFB 20090916 *)
(* NegLimitSw edges		DONE and TESTED DFB 20090916 *)

FUNCTION SMR_HomeFindEdge

(****************************************************************************************)
(* Set return value to get rid of compiler warning										*)
(****************************************************************************************)

SMR_HomeFindEdge:=	FALSE;

(****************************************************************************************)
(* Map pointer to internal homing variables 											*)
(****************************************************************************************)

t ACCESS ADR(pAxis.Internal.Homing);

(****************************************************************************************)
(* HomeSw																				*)
(****************************************************************************************)

(* Find rising and falling edges (only depends on level of switch) *)

t.RisingEdge:=	pAxis.Internal.DIGIN.HomeSw AND NOT(t.HomeSwOld);

t.FallingEdge:=	t.HomeSwOld AND NOT(pAxis.Internal.DIGIN.HomeSw);

(* Find Positive and Negative edges ( depends on direction of travel) *)

IF( t.RisingEdge ) THEN

	IF( t.CurrDirection = SMR_DIR_POS ) THEN

		t.PosEdge:=	1;
		t.NegEdge:=	0;

 	ELSIF( t.CurrDirection = SMR_DIR_NEG ) THEN

		t.PosEdge:=	0;
		t.NegEdge:=	1;

 	ELSE

		t.PosEdge:=	0;
		t.NegEdge:=	0;

	END_IF

ELSIF( t.FallingEdge ) THEN

	IF( t.CurrDirection = SMR_DIR_POS ) THEN

		t.PosEdge:=	0;
		t.NegEdge:=	1;

 	ELSIF( t.CurrDirection = SMR_DIR_NEG ) THEN

		t.PosEdge:=	1;
		t.NegEdge:=	0;

 	ELSE

		t.PosEdge:=	0;
		t.NegEdge:=	0;

	END_IF

ELSE

	t.PosEdge:=	0;
	t.NegEdge:=	0;

END_IF

(* Save value of HomeSw *)

t.HomeSwOld:=	pAxis.Internal.DIGIN.HomeSw;

(****************************************************************************************)
(* PosLimitSw																			*)
(****************************************************************************************)

(* Check for edge on PosLimitSw *)

t.PosLimitSwRisingEdge:=	pAxis.Internal.DIGIN.PosLimitSw AND NOT(t.PosLimitSwOld);

t.PosLimitSwFallingEdge:=	t.PosLimitSwOld AND NOT(pAxis.Internal.DIGIN.PosLimitSw);

(* Save value of PosLimitSw *)

t.PosLimitSwOld:=	pAxis.Internal.DIGIN.PosLimitSw;

(****************************************************************************************)
(* NegLimitSw																			*)
(****************************************************************************************)

(* Check for edge on NegLimitSw *)

t.NegLimitSwRisingEdge:=	pAxis.Internal.DIGIN.NegLimitSw AND NOT(t.NegLimitSwOld);

t.NegLimitSwFallingEdge:=	t.NegLimitSwOld AND NOT(pAxis.Internal.DIGIN.NegLimitSw);

(* Save value of PosLimitSw *)

t.NegLimitSwOld:=	pAxis.Internal.DIGIN.NegLimitSw;

END_FUNCTION

(* ---- SMR_SetBusyDone.st ---- *)
(*
* File: SMR_SetBusyDone.st
* Copyright (c) 2023 Loupe
* https://loupe.team
*
* This file is part of SMRamp, licensed under the MIT License.
*
*)

(********************************************************************)
(* Function to set Busy and Done in the ST_ENABLED state 			*)
(********************************************************************)

(* WAIT						DONE and TESTED DFB 20110405 *)
	(* No CMD				DONE and TESTED DFB 20110405 *)
	(* Home					DONE and TESTED DFB 20110405 *)
	(* MoveAbsolute			DONE and TESTED DFB 20110405 *)
	(* MoveAdditive			DONE and TESTED DFB 20110405 *)
	(* MoveVelocity			DONE and TESTED DFB 20110405 *)
	(* TrackSetPosition		DONE and TESTED DFB 20110405 *)
	(* Stop					DONE and TESTED DFB 20110405 *)
	(* Other mode			DONE and TESTED DFB 20110405 *)

(* PARWRITE					DONE and TESTED DFB 20110404 *)
(* HOME						DONE and TESTED DFB 20110404 *)
(* JOGFWD					DONE and TESTED DFB 20110419 *)
(* JOGREV					DONE and TESTED DFB 20110419 *)
(* TRACKSETPOS				DONE and TESTED DFB 20110405 *)
(* SETPOS					DONE and TESTED DFB 20110405 *)
(* SETVEL					DONE and TESTED DFB 20110405 *)
(* SETSTOP					DONE and TESTED DFB 20110405 *)
(* ERROR					DONE and TESTED DFB 20110405 *)

FUNCTION SMR_SetBusyDone

(********************************************************************)
(* Set return value to get rid of compiler warning					*)
(********************************************************************)

SMR_SetBusyDone:=	FALSE;

(********************************************************************)
(* Reset TargetReachedTimer. It is set below where needed			*)
(********************************************************************)

pAxis.Internal.TargetReachedTimer.IN:=	0;

(********************************************************************)
(* Set Busy and Done based on EnableState 							*)
(********************************************************************)

CASE pAxis.Internal.EnableState OF

	SMR_STEN_WAIT:

		(* If waiting, Busy and Done are complex *)

		(* If no commands are present, reset Busy and Done *)

		IF( 	NOT(pAxis.IN.CMD.Home)
			AND	NOT(pAxis.IN.CMD.MoveAbsolute)
			AND	NOT(pAxis.IN.CMD.MoveAdditive)
			AND	NOT(pAxis.IN.CMD.MoveVelocity)
			AND	NOT(pAxis.IN.CMD.TrackSetPosition)
			AND	NOT(pAxis.IN.CMD.Stop)
			)THEN

			pAxis.OUT.STAT.Busy:=	0;
			pAxis.OUT.STAT.Done:=	0;

		ELSE

			(* Otherwise, set Busy and Done based on MpGenMode *)

			CASE pAxis.IOMap.OUT.MpGenMode OF

				SMR_MODE_POSITION:

					(* Position mode is active for
						MoveAbsolute, MoveAdditive, Home (done homing) *)

					(* Set Busy and Done based on actual and set positions *)

					IF( pAxis.Internal.AbsPosActVal = pAxis.Internal.CurrTargetPos )THEN

		   				pAxis.OUT.STAT.Busy:=	0;
						pAxis.OUT.STAT.Done:=	1;

					ELSE

						pAxis.OUT.STAT.Busy:=	1;
						pAxis.OUT.STAT.Done:=	0;

					END_IF

				SMR_MODE_VELOCITY:

					(* Velocity mode is active for
						MoveVelocity, if a limit switch is active *)

					(* Set Busy and Done based on a TargetReached timer *)

					pAxis.Internal.TargetReachedTimer.IN:=	pAxis.OUT.STAT.DriveStatus.TargetReached;

					pAxis.OUT.STAT.Busy:=	NOT(pAxis.Internal.TargetReachedTimer.Q);
					pAxis.OUT.STAT.Done:=	pAxis.Internal.TargetReachedTimer.Q;

				ELSE

					(* These modes are active outside of this library *)

					(* Reset Busy and Done *)

					pAxis.OUT.STAT.Busy:=	0;
					pAxis.OUT.STAT.Done:=	0;

			END_CASE

		END_IF

	SMR_STEN_PARWRITE:

		(* Reset Busy to allow Par updates *)

		pAxis.OUT.STAT.Busy:=	0;
		pAxis.OUT.STAT.Done:=	0;

	SMR_STEN_HOME:

		(* If homing, Busy *)

		pAxis.OUT.STAT.Busy:=	1;
		pAxis.OUT.STAT.Done:=	0;

	SMR_STEN_JOGFWD..SMR_STEN_JOGREV:

		(* Set Busy and Done based on a TargetReached timer *)

		pAxis.Internal.TargetReachedTimer.IN:=	pAxis.OUT.STAT.DriveStatus.TargetReached;

		pAxis.OUT.STAT.Busy:=	NOT(pAxis.Internal.TargetReachedTimer.Q);
		pAxis.OUT.STAT.Done:=	pAxis.Internal.TargetReachedTimer.Q;

	SMR_STEN_TRACKSETPOS:

		(* If tracking set position, set Busy and Done based on actual and set positions *)

		IF( pAxis.Internal.AbsPosActVal = pAxis.Internal.CurrTargetPos )THEN

			pAxis.OUT.STAT.Busy:=	0;
			pAxis.OUT.STAT.Done:=	1;

		ELSE

			pAxis.OUT.STAT.Busy:=	1;
			pAxis.OUT.STAT.Done:=	0;

		END_IF

	SMR_STEN_SETPOS..SMR_STEN_SETVEL:

		(* If setting control variables, Busy *)

		pAxis.OUT.STAT.Busy:=	1;
		pAxis.OUT.STAT.Done:=	0;

	SMR_STEN_SETSTOP:

		(* If stopped, set Busy and Done based on a TargetReached timer *)

		pAxis.Internal.TargetReachedTimer.IN:=	pAxis.OUT.STAT.DriveStatus.TargetReached;

		pAxis.OUT.STAT.Busy:=	NOT(pAxis.Internal.TargetReachedTimer.Q);
		pAxis.OUT.STAT.Done:=	pAxis.Internal.TargetReachedTimer.Q;

	SMR_STEN_ERROR:

		(* If Error, reset Busy and Done *)

		pAxis.OUT.STAT.Busy:=	0;
		pAxis.OUT.STAT.Done:=	0;

END_CASE

(********************************************************************)
(* Handle TargetReachedTimer 										*)
(********************************************************************)

pAxis.Internal.TargetReachedTimer.PT:=	T#100ms;

pAxis.Internal.TargetReachedTimer();

END_FUNCTION

(* ---- SMR_SetErrorString.st ---- *)
(*
* File: SMR_SetErrorString.st
* Copyright (c) 2023 Loupe
* https://loupe.team
*
* This file is part of SMRamp, licensed under the MIT License.
*
*)

(********************************************************************)
(* Set the error string based on the error ID 						*)
(********************************************************************)

(* Functionality			DONE and TESTED DFB 20120503 *)

FUNCTION SMR_SetErrorString

(************************************************************)
(* Set return value to get rid of compile warning 			*)
(************************************************************)

SMR_SetErrorString:=	FALSE;

(* Set ErrorString *)

CASE ErrorID OF

	0:	ErrorString:=	'';

	30190..30196:	ErrorString:=	'Error writing parameters. Check IN.CFG.ModuleINADeviceName and IN.CFG.MotorIndex.';

	SMR_ERR_INVALIDPAR_ACC:		ErrorString:=	'IN.PAR.Acceleration is 0';
	SMR_ERR_INVALIDPAR_DEC:		ErrorString:=	'IN.PAR.Deceleration is 0';
	SMR_ERR_INVALIDPAR_STOPDEC:	ErrorString:=	'IN.PAR.StopDeceleration is 0';
	SMR_ERR_INVALIDPAR_DIR:		ErrorString:=	'IN.PAR.Direction is invalid';

	SMR_ERR_HOME_INVALIDPAR:	ErrorString:=	'One or more homing parameters is invalid';
	SMR_ERR_HOME_ERR:			ErrorString:=	'Error occurred while homing. Check wiring of switches and homing configuration.';

	SMR_ERR_POSLIMSW:	ErrorString:=	'Positive limit switch is active. Movement in the positive direction is not allowed.';
	SMR_ERR_NEGLIMSW:	ErrorString:=	'Negative limit switch is active. Movement in the negative direction is not allowed.';

	ELSE ErrorString:=	'Unknown error';

END_CASE

END_FUNCTION

(* ---- SMR_SetMpGenControl.st ---- *)
(*
* File: SMR_SetMpGenControl.st
* Copyright (c) 2023 Loupe
* https://loupe.team
*
* This file is part of SMRamp, licensed under the MIT License.
*
*)

(*This function sets the bits in the control word based on the axis input values.*)

(* SwOn, EnableOperation					DONE and TESTED DFB 20110906 *)
	(* Setting								see SMR_Cyclic.st *)
	(* Resetting							DONE and TESTED DFB 20110906 *)

(* VoltageEnable							DONE and TESTED DFB 20110906 *)

(* QuickStop								DONE and TESTED DFB 20110906 *)

(* FaultReset, WarningReset					DONE and TESTED DFB 20110906 *)
	(* Set									DONE and TESTED DFB 20110906 *)
	(* Reset								DONE and TESTED DFB 20110906 *)

(* UnderCurrentDetection					DONE and TESTED DFB 20110906 *)
(* ABRSynsAsync								DONE and TESTED DFB 20110906 *)
(* StallDetection							DONE and TESTED DFB 20110906 *)

FUNCTION SMR_SetMpGenControl

(********************************************************************)
(* Set return value to get rid of compiler warning					*)
(********************************************************************)

SMR_SetMpGenControl:=	FALSE;

(* Switch On and Enable Operation control bits are set in the state machine  *)
(* They are reset here *)

IF( NOT(pAxis.IN.CMD.Power) ) THEN

	pAxis.IOMap.OUT.MpGenControl:=	BIT_CLR(pAxis.IOMap.OUT.MpGenControl, SMR_CTRLBIT_SWON);
	pAxis.IOMap.OUT.MpGenControl:=	BIT_CLR(pAxis.IOMap.OUT.MpGenControl, SMR_CTRLBIT_ENABLEOPERATION);

END_IF

(* Set VoltageEnable bit always TRUE *)

pAxis.IOMap.OUT.MpGenControl:=	BIT_SET(pAxis.IOMap.OUT.MpGenControl, SMR_CTRLBIT_ENABLEVOLTAGE);

(* Set quickstop control bit accordingly *)

IF( pAxis.Internal.DIGIN.QuickStop ) THEN

	pAxis.IOMap.OUT.MpGenControl:=	BIT_SET(pAxis.IOMap.OUT.MpGenControl, SMR_CTRLBIT_QUICKSTOP);

ELSE

	pAxis.IOMap.OUT.MpGenControl:=	BIT_CLR(pAxis.IOMap.OUT.MpGenControl, SMR_CTRLBIT_QUICKSTOP);

END_IF

(* Set Fault Reset and warning reset control bits according to CMD  *)

IF( pAxis.IN.CMD.AcknowledgeError ) THEN

	(* Reset latch timer *)

	pAxis.Internal.AckResetTimer.IN:=	0;

	(* Set bits *)

	pAxis.IOMap.OUT.MpGenControl:=	BIT_SET(pAxis.IOMap.OUT.MpGenControl, SMR_CTRLBIT_FAULTRESET);
	pAxis.IOMap.OUT.MpGenControl:=	BIT_SET(pAxis.IOMap.OUT.MpGenControl, SMR_CTRLBIT_WARNINGRESET);

ELSE

	(* Set latch timer *)

	pAxis.Internal.AckResetTimer.IN:=	1;

	(* If latch timer expires, reset bits *)

	IF( pAxis.Internal.AckResetTimer.Q )THEN

		pAxis.IOMap.OUT.MpGenControl:=	BIT_CLR(pAxis.IOMap.OUT.MpGenControl, SMR_CTRLBIT_FAULTRESET);
		pAxis.IOMap.OUT.MpGenControl:=	BIT_CLR(pAxis.IOMap.OUT.MpGenControl, SMR_CTRLBIT_WARNINGRESET);

	END_IF

END_IF

(* Handle AckResetTimer *)

pAxis.Internal.AckResetTimer.PT:=	T#25ms;

pAxis.Internal.AckResetTimer();

(* Set configuration control bits according to CFG  *)

IF( pAxis.IN.CFG.UnderCurrentDetection ) THEN

	pAxis.IOMap.OUT.MpGenControl:=	BIT_SET(pAxis.IOMap.OUT.MpGenControl, SMR_CTRLBIT_UNDERCURRENT);

ELSE

	pAxis.IOMap.OUT.MpGenControl:=	BIT_CLR(pAxis.IOMap.OUT.MpGenControl, SMR_CTRLBIT_UNDERCURRENT);

END_IF

IF( pAxis.IN.CFG.ABRCtrSyncAsync ) THEN

	pAxis.IOMap.OUT.MpGenControl:=	BIT_SET(pAxis.IOMap.OUT.MpGenControl, SMR_CTRLBIT_SYNCPOS);

ELSE

	pAxis.IOMap.OUT.MpGenControl:=	BIT_CLR(pAxis.IOMap.OUT.MpGenControl, SMR_CTRLBIT_SYNCPOS);

END_IF

IF( pAxis.IN.CFG.StallDetection ) THEN

	pAxis.IOMap.OUT.MpGenControl:=	BIT_SET(pAxis.IOMap.OUT.MpGenControl, SMR_CTRLBIT_STALLDETECT);

ELSE

	pAxis.IOMap.OUT.MpGenControl:=	BIT_CLR(pAxis.IOMap.OUT.MpGenControl, SMR_CTRLBIT_STALLDETECT);

END_IF

END_FUNCTION

(* ---- SMR_SetState.st ---- *)
(*
* File: SMR_SetState.st
* Copyright (c) 2023 Loupe
* https://loupe.team
*
* This file is part of SMRamp, licensed under the MIT License.
*
*)

(*This function sets the state based on the status bits.*)

(* SMR_ST_NOTRDYTOSWON				DONE and TESTED DFB 20090909 *)
(* SMR_ST_SWONDISABLED				DONE and TESTED DFB 20090909 *)
(* SMR_ST_RDYTOSWON					DONE and TESTED DFB 20090909 *)
(* SMR_ST_SWON						DONE and TESTED DFB 20090909 *)
(* SMR_ST_ENABLED					DONE and TESTED DFB 20090909 *)
(* SMR_ST_QUICKSTOPACTIVE			DONE and TESTED DFB 20090909 *)
(* SMR_ST_FAULTRXNACTIVE			DONE and TESTED DFB 20090909 *)
(* SMR_ST_FAULT						DONE and TESTED DFB 20090909 *)

FUNCTION SMR_SetState

(********************************************************************)
(* Set return value to get rid of compiler warning					*)
(********************************************************************)

SMR_SetState:=	FALSE;

(* Set state *)

IF( 	(t.DriveStatus.RdyToSwOn = 0)
	AND	(t.DriveStatus.SwOn = 0)
	AND	(t.DriveStatus.OpEnabled = 0)
 	AND	(t.DriveStatus.Fault = 0)
	AND	(t.DriveStatus.SwOnDisabled = 0)
	)THEN

	t.State:=	SMR_ST_NOTRDYTOSWON;

ELSIF(		(t.DriveStatus.RdyToSwOn = 0)
		AND (t.DriveStatus.SwOn = 0)
		AND	(t.DriveStatus.OpEnabled = 0)
		AND	(t.DriveStatus.Fault = 0)
		AND	(t.DriveStatus.SwOnDisabled = 1)
		)THEN

	t.State:=	SMR_ST_SWONDISABLED;

ELSIF(		(t.DriveStatus.RdyToSwOn = 1)
		AND	(t.DriveStatus.SwOn = 0)
		AND	(t.DriveStatus.OpEnabled = 0)
		AND	(t.DriveStatus.Fault = 0)
		AND	(t.DriveStatus.QuickStop = 1)
  		AND	(t.DriveStatus.SwOnDisabled = 0)
		)THEN

	t.State:=	SMR_ST_RDYTOSWON;

ELSIF(		(t.DriveStatus.RdyToSwOn = 1)
		AND	(t.DriveStatus.SwOn = 1)
		AND	(t.DriveStatus.OpEnabled = 0)
		AND	(t.DriveStatus.Fault = 0)
		AND	(t.DriveStatus.QuickStop = 1)
		AND	(t.DriveStatus.SwOnDisabled = 0)
		)THEN

	t.State:=	SMR_ST_SWON;

ELSIF(		(t.DriveStatus.RdyToSwOn = 1)
		AND	(t.DriveStatus.SwOn = 1)
		AND	(t.DriveStatus.OpEnabled = 1)
		AND	(t.DriveStatus.Fault = 0)
  		AND	(t.DriveStatus.QuickStop = 1)
		AND	(t.DriveStatus.SwOnDisabled = 0)
		)THEN

	t.State:=	SMR_ST_ENABLED;

ELSIF(		(t.DriveStatus.RdyToSwOn = 1)
		AND	(t.DriveStatus.SwOn = 1)
		AND	(t.DriveStatus.OpEnabled = 1)
		AND	(t.DriveStatus.Fault = 0)
		AND	(t.DriveStatus.QuickStop = 0)
		AND	(t.DriveStatus.SwOnDisabled = 0)
		)THEN

	t.State:=	SMR_ST_QUICKSTOPACTIVE;

ELSIF(		(t.DriveStatus.RdyToSwOn = 1)
		AND	(t.DriveStatus.SwOn = 1)
		AND	(t.DriveStatus.OpEnabled = 1)
		AND	(t.DriveStatus.Fault = 1)
		AND	(t.DriveStatus.SwOnDisabled = 0)
		)THEN

	t.State:=	SMR_ST_FAULTRXNACTIVE;

ELSIF(		(t.DriveStatus.RdyToSwOn = 0)
		AND	(t.DriveStatus.SwOn = 0)
		AND	(t.DriveStatus.OpEnabled = 0)
		AND	(t.DriveStatus.Fault = 1)
		AND	(t.DriveStatus.SwOnDisabled = 0)
		)THEN

	t.State:=	SMR_ST_FAULT;

END_IF

END_FUNCTION

(* ---- SMR_StartHome.st ---- *)
(*
* File: SMR_StartHome.st
* Copyright (c) 2023 Loupe
* https://loupe.team
*
* This file is part of SMRamp, licensed under the MIT License.
*
*)

(********************************************************************)
(* Start a homing move 												*)
(********************************************************************)

FUNCTION SMR_StartHome

(********************************************************************)
(* Set return value to get rid of compiler warning					*)
(********************************************************************)

SMR_StartHome:=	FALSE;

(* Set Internal.CMD *)

pAxis.Internal.CMD.Home:=	1;

(* Set Invalid Direction to disable default limit switch monitoring *)
(* Limit switches are monitored inside of the homing procedure *)

pAxis.Internal.CurrDirection:=	SMR_DIR_INVALID;

(* Reset HomingOk *)

pAxis.OUT.STAT.DriveStatus.HomingOk:=	0;

(* Initialize Homing variables *)

pAxis.Internal.Homing.State:=			SMR_STHOME_CHECKMODE;
pAxis.Internal.Homing.CurrDirection:=	SMR_DIR_STOP;
pAxis.Internal.Homing.HomeSwOld:=		pAxis.Internal.DIGIN.HomeSw;
pAxis.Internal.Homing.PosLimitSwOld:=	pAxis.Internal.DIGIN.PosLimitSw;
pAxis.Internal.Homing.NegLimitSwOld:=	pAxis.Internal.DIGIN.NegLimitSw;

(* SetState should be SMR_STEN_HOME *)

pAxis.Internal.SetState:=	SMR_STEN_HOME;

(* Check for ParsOK *)

IF( pAxis.Internal.ParsOK ) THEN

	pAxis.Internal.EnableState:=	pAxis.Internal.SetState;

ELSE

	pAxis.Internal.EnableState:=	SMR_STEN_PARWRITE;

END_IF

END_FUNCTION

(* ---- SMR_StartJogForward.st ---- *)
(*
* File: SMR_StartJogForward.st
* Copyright (c) 2023 Loupe
* https://loupe.team
*
* This file is part of SMRamp, licensed under the MIT License.
*
*)

(********************************************************************)
(* Starts a JogForward move 										*)
(********************************************************************)

FUNCTION SMR_StartJogForward

(********************************************************************)
(* Set return value to get rid of compiler warning					*)
(********************************************************************)

SMR_StartJogForward:=	FALSE;

(* Set Internal.CMD *)

pAxis.Internal.CMD.JogForward:=	1;

(* Set the target state as SMR_STEN_JOGFWD *)

pAxis.Internal.SetState:=		SMR_STEN_JOGFWD;

(* Check for ParsOK *)

IF( pAxis.Internal.ParsOK ) THEN

	pAxis.Internal.EnableState:=	pAxis.Internal.SetState;

ELSE

	pAxis.Internal.EnableState:=	SMR_STEN_PARWRITE;

END_IF

(* Set CurrTargetVel *)

pAxis.Internal.CurrTargetVel:=	pAxis.IN.PAR.JogVelocity;
pAxis.Internal.CurrDirection:=	SMR_DIR_POS;

END_FUNCTION

(* ---- SMR_StartJogReverse.st ---- *)
(*
* File: SMR_StartJogReverse.st
* Copyright (c) 2023 Loupe
* https://loupe.team
*
* This file is part of SMRamp, licensed under the MIT License.
*
*)

(********************************************************************)
(* Starts a JogReverse move 										*)
(********************************************************************)

FUNCTION SMR_StartJogReverse

(********************************************************************)
(* Set return value to get rid of compiler warning					*)
(********************************************************************)

SMR_StartJogReverse:=	FALSE;

(* Set Internal.CMD *)

pAxis.Internal.CMD.JogReverse:=	1;

(* Set the target state as SMR_STEN_JOGREV *)

pAxis.Internal.SetState:=		SMR_STEN_JOGREV;

(* Check for ParsOK *)

IF( pAxis.Internal.ParsOK ) THEN

	pAxis.Internal.EnableState:=	pAxis.Internal.SetState;

ELSE

	pAxis.Internal.EnableState:=	SMR_STEN_PARWRITE;

END_IF

(* Set CurrTargetVel *)

pAxis.Internal.CurrTargetVel:=	-1 * UINT_TO_DINT( pAxis.IN.PAR.JogVelocity );
pAxis.Internal.CurrDirection:=	SMR_DIR_NEG;

END_FUNCTION

(* ---- SMR_StartMoveAbsolute.st ---- *)
(*
* File: SMR_StartMoveAbsolute.st
* Copyright (c) 2023 Loupe
* https://loupe.team
*
* This file is part of SMRamp, licensed under the MIT License.
*
*)

(********************************************************************)
(* Start an absolute move 											*)
(********************************************************************)

FUNCTION SMR_StartMoveAbsolute

(********************************************************************)
(* Set return value to get rid of compiler warning					*)
(********************************************************************)

SMR_StartMoveAbsolute:=	FALSE;

(* Set Internal.CMD *)

pAxis.Internal.CMD.MoveAbsolute:=	1;

(* Set CurrTargetPos to input position for absolute moves *)

pAxis.Internal.CurrTargetPos:=	pAxis.IN.PAR.Position;

(* Set CurrDirection based on internal position and target position *)

IF( pAxis.Internal.CurrTargetPos > pAxis.Internal.AbsPosActVal ) THEN

	pAxis.Internal.CurrDirection:=	SMR_DIR_POS;

ELSIF( pAxis.Internal.CurrTargetPos < pAxis.Internal.AbsPosActVal ) THEN

	pAxis.Internal.CurrDirection:=	SMR_DIR_NEG;

ELSE

	pAxis.Internal.CurrDirection:=	SMR_DIR_STOP;

END_IF

(* Set the target state as SETPOS *)

pAxis.Internal.SetState:=		SMR_STEN_SETPOS;

(* Check for ParsOK *)

IF( pAxis.Internal.ParsOK ) THEN

	pAxis.Internal.EnableState:=	pAxis.Internal.SetState;

ELSE

	pAxis.Internal.EnableState:=	SMR_STEN_PARWRITE;

END_IF

END_FUNCTION

(* ---- SMR_StartMoveAdditive.st ---- *)
(*
* File: SMR_StartMoveAdditive.st
* Copyright (c) 2023 Loupe
* https://loupe.team
*
* This file is part of SMRamp, licensed under the MIT License.
*
*)

(********************************************************************)
(* Start an additive move 											*)
(********************************************************************)

FUNCTION SMR_StartMoveAdditive

(********************************************************************)
(* Set return value to get rid of compiler warning					*)
(********************************************************************)

SMR_StartMoveAdditive:=	FALSE;

(* Set Internal.CMD *)

pAxis.Internal.CMD.MoveAdditive:=	1;

(* For additive moves, CurrTargetPos depends on current motion mode *)

IF( pAxis.IOMap.OUT.MpGenMode = SMR_MODE_POSITION ) THEN

	(* Add input position to CurrTargetPos if already in position mode *)

	pAxis.Internal.CurrTargetPos:=	pAxis.Internal.CurrTargetPos + pAxis.IN.PAR.Position;

ELSIF( pAxis.IOMap.OUT.MpGenMode = SMR_MODE_VELOCITY ) THEN

	(* If currently in velocity mode, add input position to current position *)

	pAxis.Internal.CurrTargetPos:=	pAxis.Internal.AbsPosActVal + pAxis.IN.PAR.Position;

(* WHAT ABOUT OTHER MODES??? *)

END_IF

(* Set CurrDirection based on internal position and target position *)

IF( pAxis.Internal.CurrTargetPos > pAxis.Internal.AbsPosActVal ) THEN

	pAxis.Internal.CurrDirection:=	SMR_DIR_POS;

ELSIF( pAxis.Internal.CurrTargetPos < pAxis.Internal.AbsPosActVal ) THEN

	pAxis.Internal.CurrDirection:=	SMR_DIR_NEG;

ELSE

	pAxis.Internal.CurrDirection:=	SMR_DIR_STOP;

END_IF

(* Set the target state as SETPOS *)

pAxis.Internal.SetState:=		SMR_STEN_SETPOS;

(* Check for ParsOK *)

IF( pAxis.Internal.ParsOK ) THEN

	pAxis.Internal.EnableState:=	pAxis.Internal.SetState;

ELSE

	pAxis.Internal.EnableState:=	SMR_STEN_PARWRITE;

END_IF

END_FUNCTION

(* ---- SMR_StartMoveVelocity.st ---- *)
(*
* File: SMR_StartMoveVelocity.st
* Copyright (c) 2023 Loupe
* https://loupe.team
*
* This file is part of SMRamp, licensed under the MIT License.
*
*)

(********************************************************************)
(* Start a velocity move 											*)
(********************************************************************)

FUNCTION SMR_StartMoveVelocity

(********************************************************************)
(* Set return value to get rid of compiler warning					*)
(********************************************************************)

SMR_StartMoveVelocity:=	FALSE;

(* Set Internal.CMD *)

pAxis.Internal.CMD.MoveVelocity:=	1;

(* These conditionals have a different order than MoveAdditive and MoveAbsolute.
	This is because of the error checking on direction.
	If there is a direction error, then the error state transition
	needs to override any other state transition.
	So, the direction check needs to happen after the parameter checks *)

(* Set the target state as SETVEL *)

pAxis.Internal.SetState:=		SMR_STEN_SETVEL;

(* Check for ParsOK *)

IF( pAxis.Internal.ParsOK ) THEN

	pAxis.Internal.EnableState:=	pAxis.Internal.SetState;

ELSE

	pAxis.Internal.EnableState:=	SMR_STEN_PARWRITE;

END_IF

(* Set CurrTargetVel based on input velocity and direction *)

IF( pAxis.IN.PAR.Direction = SMR_DIR_POS ) THEN

	pAxis.Internal.CurrTargetVel:=	pAxis.IN.PAR.Velocity;
	pAxis.Internal.CurrDirection:=	SMR_DIR_POS;

ELSIF( pAxis.IN.PAR.Direction = SMR_DIR_NEG ) THEN

	pAxis.Internal.CurrTargetVel:=	-1 * UINT_TO_DINT(pAxis.IN.PAR.Velocity);
	pAxis.Internal.CurrDirection:=	SMR_DIR_NEG;

ELSE

	(* Invalid direction - Grab error info and abort move *)

	pAxis.Internal.Error:=			1;
	pAxis.OUT.STAT.ErrorID:=		SMR_ERR_INVALIDPAR_DIR;
	pAxis.OUT.STAT.ErrorState:=		SMR_STEN_WAIT;

	pAxis.Internal.EnableState:=	SMR_STEN_ERROR;

END_IF

END_FUNCTION

(* ---- SMR_StartTrackSetPosition.st ---- *)
(*
* File: SMR_StartTrackSetPosition.st
* Copyright (c) 2023 Loupe
* https://loupe.team
*
* This file is part of SMRamp, licensed under the MIT License.
*
*)

(********************************************************************)
(* Starts a TrackSetPosition move 									*)
(********************************************************************)

FUNCTION SMR_StartTrackSetPosition

(********************************************************************)
(* Set return value to get rid of compiler warning					*)
(********************************************************************)

SMR_StartTrackSetPosition:=	FALSE;

(* Set Internal.CMD *)

pAxis.Internal.CMD.TrackSetPosition:=	1;

(* Set CurrTargetPos to input position for absolute moves *)

pAxis.Internal.CurrTargetPos:=	pAxis.IN.PAR.Position;

(* Set CurrDirection based on internal position and target position *)

IF( pAxis.Internal.CurrTargetPos > pAxis.Internal.AbsPosActVal ) THEN

	pAxis.Internal.CurrDirection:=	SMR_DIR_POS;

ELSIF( pAxis.Internal.CurrTargetPos < pAxis.Internal.AbsPosActVal ) THEN

	pAxis.Internal.CurrDirection:=	SMR_DIR_NEG;

ELSE

	pAxis.Internal.CurrDirection:=	SMR_DIR_STOP;

END_IF

(* Set the target state as TRACKSETPOS *)

pAxis.Internal.SetState:=		SMR_STEN_TRACKSETPOS;

(* Check for ParsOK *)

IF( pAxis.Internal.ParsOK ) THEN

	pAxis.Internal.EnableState:=	pAxis.Internal.SetState;

ELSE

	pAxis.Internal.EnableState:=	SMR_STEN_PARWRITE;

END_IF

END_FUNCTION

(* ---- SMR_UpdatePars.st ---- *)
(*
* File: SMR_UpdatePars.st
* Copyright (c) 2023 Loupe
* https://loupe.team
*
* This file is part of SMRamp, licensed under the MIT License.
*
*)

(********************************************************************)
(* Update motion parameters if they change	 						*)
(********************************************************************)

(* Disable Acyclic Write			DONE and TESTED DFB 20110404 *)
	(* Disable FUBs					DONE and TESTED DFB 20110404 *)
	(* Set ParsOK					DONE and TESTED DFB 20110404 *)
	(* Return						DONE and TESTED DFB 20110404 *)

(* Checking invalid pars			DONE and TESTED DFB 20110404 *)
	(* Accel						DONE and TESTED DFB 20110404 *)
	(* Decel						DONE and TESTED DFB 20110404 *)
	(* StopDecel					DONE and TESTED DFB 20110404 *)

(* Update Velocity					DONE and TESTED DFB 20110404 *)

	(* Check for changes			DONE and TESTED DFB 20110404 *)
		(* DisAccWrite transition	DONE and TESTED DFB 20110404 *)
		(* Busy						DONE and TESTED DFB 20110404 *)
		(* Error					DONE and TESTED DFB 20110404 *)
		(* Not Busy or Error		DONE and TESTED DFB 20110404 *)

	(* AccWrite						DONE and TESTED DFB 20110404 *)
		(* FUB done					DONE and TESTED DFB 20110404 *)
		(* No Error					DONE and TESTED DFB 20110404 *)
		(* Error					DONE and TESTED DFB 20110404 *)

(* Update Acceleration				DONE and TESTED DFB 20110404 *)

	(* Check for changes			DONE and TESTED DFB 20110404 *)
		(* DisAccWrite transition	DONE and TESTED DFB 20110404 *)
		(* Busy						DONE and TESTED DFB 20110404 *)
		(* Error					DONE and TESTED DFB 20110404 *)
		(* Not Busy or Error		DONE and TESTED DFB 20110404 *)

	(* AccWrite						DONE and TESTED DFB 20110404 *)
		(* FUB done					DONE and TESTED DFB 20110404 *)
		(* No Error					DONE and TESTED DFB 20110404 *)
		(* Error					DONE and TESTED DFB 20110404 *)

(* Update Deceleration				DONE and TESTED DFB 20110404 *)

	(* Check for changes			DONE and TESTED DFB 20110404 *)
		(* DisAccWrite transition	DONE and TESTED DFB 20110404 *)
		(* Stopping					DONE and TESTED DFB 20110404 *)
			(* Busy					DONE and TESTED DFB 20110404 *)
			(* Error				DONE and TESTED DFB 20110404 *)
			(* Not Busy or Error	DONE and TESTED DFB 20110404 *)
		(* Not stopping				DONE and TESTED DFB 20110404 *)
			(* Busy					DONE and TESTED DFB 20110404 *)
			(* Error				DONE and TESTED DFB 20110404 *)
			(* Not Busy or Error	DONE and TESTED DFB 20110404 *)

	(* AccWrite						DONE and TESTED DFB 20110404 *)
		(* Proper decel value		DONE and TESTED DFB 20110404 *)
			(* Stopping				DONE and TESTED DFB 20110404 *)
			(* Not stopping			DONE and TESTED DFB 20110404 *)
		(* FUB done					DONE and TESTED DFB 20110404 *)
		(* No Error					DONE and TESTED DFB 20110404 *)
		(* Error					DONE and TESTED DFB 20110404 *)

(* Setting ParsOK					DONE and TESTED DFB 20110404 *)

FUNCTION SMR_UpdatePars

(********************************************************************)
(* Set return value to get rid of compiler warning					*)
(********************************************************************)

SMR_UpdatePars:=	FALSE;

(********************************************************************)
(* Check DisableAcyclicWrite										*)
(********************************************************************)

IF( pAxis.IN.CFG.DisableAcyclicWrite )THEN

	(* Disable FUBs *)

	pAxis.Internal.UpdateVel.AccWrite.enable:=	0;
	pAxis.Internal.UpdateAcc.AccWrite.enable:=	0;
	pAxis.Internal.UpdateDec.AccWrite.enable:=	0;

	(* Set ParsOK *)

	pAxis.Internal.ParsOK:=	1;

	(* Return *)

	RETURN;

END_IF

(********************************************************************)
(* Check Accel and Decel PARs										*)
(********************************************************************)

IF( pAxis.IN.PAR.Acceleration = 0 ) THEN

	(* Disable FUBs *)

	pAxis.Internal.UpdateVel.AccWrite.enable:=	0;
	pAxis.Internal.UpdateAcc.AccWrite.enable:=	0;
	pAxis.Internal.UpdateDec.AccWrite.enable:=	0;

	(* Grab error info *)

	pAxis.Internal.Error:=			1;
	pAxis.OUT.STAT.ErrorID:=		SMR_ERR_INVALIDPAR_ACC;
	pAxis.OUT.STAT.ErrorState:=		pAxis.Internal.EnableState;

	pAxis.Internal.EnableState:=	SMR_STEN_ERROR;

	(* Reset ParsOK *)

	pAxis.Internal.ParsOK:=	0;

	(* Return *)

	RETURN;

END_IF

IF( pAxis.IN.PAR.Deceleration = 0 ) THEN

	(* Disable FUBs *)

	pAxis.Internal.UpdateVel.AccWrite.enable:=	0;
	pAxis.Internal.UpdateAcc.AccWrite.enable:=	0;
	pAxis.Internal.UpdateDec.AccWrite.enable:=	0;

	(* Grab error info *)

	pAxis.Internal.Error:=			1;
	pAxis.OUT.STAT.ErrorID:=		SMR_ERR_INVALIDPAR_DEC;
	pAxis.OUT.STAT.ErrorState:=		pAxis.Internal.EnableState;

	pAxis.Internal.EnableState:=	SMR_STEN_ERROR;

	(* Reset ParsOK *)

	pAxis.Internal.ParsOK:=	0;

	(* Return *)

	RETURN;

END_IF

IF( pAxis.IN.PAR.StopDeceleration = 0 ) THEN

	(* Disable FUBs *)

	pAxis.Internal.UpdateVel.AccWrite.enable:=	0;
	pAxis.Internal.UpdateAcc.AccWrite.enable:=	0;
	pAxis.Internal.UpdateDec.AccWrite.enable:=	0;

	(* Grab error info *)

	pAxis.Internal.Error:=			1;
	pAxis.OUT.STAT.ErrorID:=		SMR_ERR_INVALIDPAR_STOPDEC;
	pAxis.OUT.STAT.ErrorState:=		pAxis.Internal.EnableState;

	pAxis.Internal.EnableState:=	SMR_STEN_ERROR;

	(* Reset ParsOK *)

	pAxis.Internal.ParsOK:=	0;

	(* Return *)

	RETURN;

END_IF

(********************************************************************)
(* Velocity															*)
(********************************************************************)

IF( (pAxis.IN.PAR.Velocity <> pAxis.Internal.UpdateVel.CurrValue)
	AND NOT(pAxis.OUT.STAT.Busy)
	AND NOT(pAxis.OUT.STAT.Error)
	)THEN

	pAxis.Internal.UpdateVel.Update:=	1;

END_IF

IF( pAxis.Internal.UpdateVel.Update )THEN

	(* Handle Acyclic write *)

	pAxis.Internal.UpdateVel.AccWrite.enable:=		1;
	pAxis.Internal.UpdateVel.AccWrite.pDeviceName:=	ADR(pAxis.IN.CFG.ModuleINADeviceName);

	(* Set channel name based on motor index *)

	CASE pAxis.IN.CFG.MotorIndex OF

		1:		pAxis.Internal.UpdateVel.AccWrite.pChannelName:=	ADR('MaxSpeed01pos');
		2:		pAxis.Internal.UpdateVel.AccWrite.pChannelName:=	ADR('MaxSpeed02pos');
		3:		pAxis.Internal.UpdateVel.AccWrite.pChannelName:=	ADR('MaxSpeed03pos');
		4:		pAxis.Internal.UpdateVel.AccWrite.pChannelName:=	ADR('MaxSpeed04pos');
		ELSE	pAxis.Internal.UpdateVel.AccWrite.pChannelName:=	ADR('badname');

	END_CASE

	pAxis.Internal.UpdateVel.AccWrite.value:=	pAxis.IN.PAR.Velocity;

	(* Check Status *)

	IF( pAxis.Internal.UpdateVel.AccWrite.status < SMR_STAT_DISABLED ) THEN

		(* FUB finished, disable *)

		pAxis.Internal.UpdateVel.AccWrite.enable:=	0;

		(* Reset CMD *)

		pAxis.Internal.UpdateVel.Update:=	0;

		(* Check for error *)

		IF( pAxis.Internal.UpdateVel.AccWrite.status = 0 ) THEN

			(* Set CurrValue to input *)

			pAxis.Internal.UpdateVel.CurrValue:=	UDINT_TO_UINT(pAxis.Internal.UpdateVel.AccWrite.value);

		ELSE

			(* Grab error info and go to error state *)

			pAxis.Internal.Error:=			1;
			pAxis.OUT.STAT.Error:=			1;
			pAxis.OUT.STAT.ErrorID:=		pAxis.Internal.UpdateVel.AccWrite.status;
			pAxis.OUT.STAT.ErrorState:=		pAxis.Internal.EnableState;

			pAxis.Internal.EnableState:=	SMR_STEN_ERROR;

		END_IF (* Status check *)

	END_IF (* FUB finished *)

END_IF (* Update *)

(********************************************************************)
(* Acceleration														*)
(********************************************************************)

IF( (pAxis.IN.PAR.Acceleration <> pAxis.Internal.UpdateAcc.CurrValue)
	AND NOT(pAxis.OUT.STAT.Busy)
	AND NOT(pAxis.OUT.STAT.Error)
	)THEN

	pAxis.Internal.UpdateAcc.Update:=	1;

END_IF

IF( pAxis.Internal.UpdateAcc.Update )THEN

	(* Handle Acyclic write *)

	pAxis.Internal.UpdateAcc.AccWrite.enable:=		1;
	pAxis.Internal.UpdateAcc.AccWrite.pDeviceName:=	ADR(pAxis.IN.CFG.ModuleINADeviceName);

	(* Set channel name based on motor index *)

	CASE pAxis.IN.CFG.MotorIndex OF

		1:		pAxis.Internal.UpdateAcc.AccWrite.pChannelName:=	ADR('MaxAcc01');
		2:		pAxis.Internal.UpdateAcc.AccWrite.pChannelName:=	ADR('MaxAcc02');
		3:		pAxis.Internal.UpdateAcc.AccWrite.pChannelName:=	ADR('MaxAcc03');
		4:		pAxis.Internal.UpdateAcc.AccWrite.pChannelName:=	ADR('MaxAcc04');
		ELSE	pAxis.Internal.UpdateAcc.AccWrite.pChannelName:=	ADR('badname');

	END_CASE

	pAxis.Internal.UpdateAcc.AccWrite.value:=	pAxis.IN.PAR.Acceleration;

	(* Check Status *)

	IF( pAxis.Internal.UpdateAcc.AccWrite.status < SMR_STAT_DISABLED ) THEN

		(* FUB finished, disable *)

		pAxis.Internal.UpdateAcc.AccWrite.enable:=	0;

		(* Reset CMD *)

		pAxis.Internal.UpdateAcc.Update:=	0;

		(* Check for error *)

		IF( pAxis.Internal.UpdateAcc.AccWrite.status = 0 ) THEN

			(* Set CurrValue to input *)

			pAxis.Internal.UpdateAcc.CurrValue:=	UDINT_TO_UINT(pAxis.Internal.UpdateAcc.AccWrite.value);

		ELSE

			(* Grab error info and go to error state *)

			pAxis.Internal.Error:=			1;
			pAxis.OUT.STAT.Error:=			1;
			pAxis.OUT.STAT.ErrorID:=		pAxis.Internal.UpdateAcc.AccWrite.status;
			pAxis.OUT.STAT.ErrorState:=		pAxis.Internal.EnableState;

			pAxis.Internal.EnableState:=	SMR_STEN_ERROR;

		END_IF (* Status check *)

	END_IF (* FUB finished *)

END_IF (* Update CMD *)

(********************************************************************)
(* Deceleration														*)
(********************************************************************)

(* Parameter checking is different for Stop condition and normal operation *)

IF( pAxis.IN.CMD.Stop )THEN

	IF( (pAxis.IN.PAR.StopDeceleration <> pAxis.Internal.UpdateDec.CurrValue)
		AND NOT(pAxis.OUT.STAT.Error)
		)THEN

		pAxis.Internal.UpdateDec.Update:=	1;

	END_IF

ELSE

	IF( (pAxis.IN.PAR.Deceleration <> pAxis.Internal.UpdateDec.CurrValue)
		AND NOT(pAxis.OUT.STAT.Busy)
		AND NOT(pAxis.OUT.STAT.Error)
		)THEN

		pAxis.Internal.UpdateDec.Update:=	1;

	END_IF

END_IF

IF( pAxis.Internal.UpdateDec.Update )THEN

	(* Handle Acyclic write *)

	pAxis.Internal.UpdateDec.AccWrite.enable:=		1;
	pAxis.Internal.UpdateDec.AccWrite.pDeviceName:=	ADR(pAxis.IN.CFG.ModuleINADeviceName);

	(* Set channel name based on motor index *)

	CASE pAxis.IN.CFG.MotorIndex OF

		1:		pAxis.Internal.UpdateDec.AccWrite.pChannelName:=	ADR('MaxDec01');
		2:		pAxis.Internal.UpdateDec.AccWrite.pChannelName:=	ADR('MaxDec02');
		3:		pAxis.Internal.UpdateDec.AccWrite.pChannelName:=	ADR('MaxDec03');
		4:		pAxis.Internal.UpdateDec.AccWrite.pChannelName:=	ADR('MaxDec04');
		ELSE	pAxis.Internal.UpdateDec.AccWrite.pChannelName:=	ADR('badname');

	END_CASE

	IF( pAxis.IN.CMD.Stop )THEN

		pAxis.Internal.UpdateDec.AccWrite.value:=	pAxis.IN.PAR.StopDeceleration;

	ELSE

		pAxis.Internal.UpdateDec.AccWrite.value:=	pAxis.IN.PAR.Deceleration;

	END_IF

	(* Check Status *)

	IF( pAxis.Internal.UpdateDec.AccWrite.status < SMR_STAT_DISABLED ) THEN

		(* FUB finished, disable *)

		pAxis.Internal.UpdateDec.AccWrite.enable:=	0;

		(* Reset CMD *)

		pAxis.Internal.UpdateDec.Update:=	0;

		(* Check for error *)

		IF( pAxis.Internal.UpdateDec.AccWrite.status = 0 ) THEN

			(* Set CurrValue to input *)

			pAxis.Internal.UpdateDec.CurrValue:=	UDINT_TO_UINT(pAxis.Internal.UpdateDec.AccWrite.value);

		ELSE

			(* Grab error info and go to error state *)

			pAxis.Internal.Error:=			1;
			pAxis.OUT.STAT.Error:=			1;
			pAxis.OUT.STAT.ErrorID:=		pAxis.Internal.UpdateDec.AccWrite.status;
			pAxis.OUT.STAT.ErrorState:=		pAxis.Internal.EnableState;

			pAxis.Internal.EnableState:=	SMR_STEN_ERROR;

		END_IF (* Status check *)

	END_IF (* FUB finished *)

END_IF (* Update CMD *)

(********************************************************************)
(* Set ParsOK appropriately											*)
(********************************************************************)

(* ParsOK is not checked on a stop condition, so, it does not need to depend on the Stop CMD
	or the StopDeceleration *)

IF( 	(pAxis.Internal.UpdateVel.CurrValue = pAxis.IN.PAR.Velocity)
	AND (pAxis.Internal.UpdateAcc.CurrValue = pAxis.IN.PAR.Acceleration)
	AND (pAxis.Internal.UpdateDec.CurrValue = pAxis.IN.PAR.Deceleration)
	)THEN

	pAxis.Internal.ParsOK:=	1;

ELSE

	pAxis.Internal.ParsOK:=	0;

END_IF

END_FUNCTION

(* ---- SMRamp.fun ---- *)
(*
* File: SMRamp.fun
* Copyright (c) 2023 Loupe
* https://loupe.team
*
* This file is part of SMRamp, licensed under the MIT License.
*
*)

FUNCTION SMR_AxisFn_Cyclic : BOOL (*This function handles cyclic motion on the Ramp Mode axis.*)
	VAR_IN_OUT
		pAxis : SMR_Axis_typ; (*SMRamp Axis object*)
	END_VAR
END_FUNCTION

FUNCTION SMR_SetMpGenControl : BOOL (*This function sets the bits in the control word based on the axis input values*)
	VAR_IN_OUT
		pAxis : SMR_Axis_typ; (*SMRamp Axis object*)
	END_VAR
END_FUNCTION

FUNCTION SMR_GetDriveStatus : BOOL (*This is an internal function that maps out the status from the status UINT*)
	VAR_INPUT
		MpGenStatus : UINT; (*MpGenStatus input*)
	END_VAR
	VAR_IN_OUT
		DriveStatus : SMR_Axis_OUT_STAT_DriveStat_typ; (*Drive status structure*)
	END_VAR
END_FUNCTION

FUNCTION SMR_SetState : BOOL (*This function sets the state based on the status bits*)
	VAR_IN_OUT
		t : SMR_Axis_OUT_STAT_typ; (*Pointer to the Output Status*)
	END_VAR
END_FUNCTION

FUNCTION SMR_Home : BOOL (*Function to perform homing functionality*)
	VAR_IN_OUT
		pAxis : SMR_Axis_typ; (*SMRamp Axis object*)
	END_VAR
	VAR
		t : REFERENCE TO SMR_Axis_Int_Homing_typ; (*Pointer to the homing variables*)
	END_VAR
END_FUNCTION

FUNCTION SMR_HomeFindEdge : BOOL (*Function to find edges for homing*)
	VAR_IN_OUT
		pAxis : SMR_Axis_typ; (*SMRamp Axis object*)
	END_VAR
	VAR
		t : REFERENCE TO SMR_Axis_Int_Homing_typ; (*Pointer to the homing variables*)
	END_VAR
END_FUNCTION

FUNCTION SMR_CheckHomePAR : BOOL (*Function which checks homing parameters.  Returns TRUE if pars are OK.*)
	VAR_IN_OUT
		pAxis : SMR_Axis_typ; (*SMRamp Axis object*)
	END_VAR
	VAR
		Error : BOOL; (*Error exists with a homing parameter*)
	END_VAR
END_FUNCTION

FUNCTION SMR_StartHome : BOOL (*Start a homing move*)
	VAR_IN_OUT
		pAxis : SMR_Axis_typ; (*SMRamp Axis object*)
	END_VAR
END_FUNCTION

FUNCTION SMR_StartMoveAbsolute : BOOL (*Start an absolute move*)
	VAR_IN_OUT
		pAxis : SMR_Axis_typ; (*SMRamp Axis object*)
	END_VAR
END_FUNCTION

FUNCTION SMR_StartMoveAdditive : BOOL (*Start an additive move*)
	VAR_IN_OUT
		pAxis : SMR_Axis_typ; (*SMRamp Axis object*)
	END_VAR
END_FUNCTION

FUNCTION SMR_StartMoveVelocity : BOOL (*Start a velocity move*)
	VAR_IN_OUT
		pAxis : SMR_Axis_typ; (*SMRamp Axis object*)
	END_VAR
END_FUNCTION

FUNCTION SMR_StartTrackSetPosition : BOOL (*Starts a TrackSetPosition move*)
	VAR_IN_OUT
		pAxis : SMR_Axis_typ; (*SMRamp Axis object*)
	END_VAR
END_FUNCTION

FUNCTION SMR_StartJogForward : BOOL (*Starts a JogForward move*)
	VAR_IN_OUT
		pAxis : SMR_Axis_typ; (*SMRamp Axis object*)
	END_VAR
END_FUNCTION

FUNCTION SMR_StartJogReverse : BOOL (*Starts a JogReverse move*)
	VAR_IN_OUT
		pAxis : SMR_Axis_typ; (*SMRamp Axis object*)
	END_VAR
END_FUNCTION

FUNCTION SMR_SetBusyDone : BOOL (*Function to set Busy and Done in the ST_ENABLED state*)
	VAR_IN_OUT
		pAxis : SMR_Axis_typ; (*SMRamp Axis object*)
	END_VAR
END_FUNCTION

FUNCTION SMR_CheckLimitSw : BOOL (*Check limit switches*)
	VAR_IN_OUT
		pAxis : SMR_Axis_typ; (*SMRamp Axis object*)
	END_VAR
END_FUNCTION

FUNCTION SMR_UpdatePars : BOOL (*Update motion parameters if they change*)
	VAR_IN_OUT
		pAxis : SMR_Axis_typ; (*SMRamp Axis object*)
	END_VAR
END_FUNCTION

FUNCTION SMR_SetErrorString : BOOL (*Set the error string based on the error ID*)
	VAR_INPUT
		ErrorID : UINT;
	END_VAR
	VAR_IN_OUT
		ErrorString : STRING[SMR_STRLEN_ERROR];
	END_VAR
END_FUNCTION
